// TwinCAT 3 PLC project PLC1
// ProgramVersion: 3.1.4026.23
// libraries:
//   Tc2_EtherCAT, * (Beckhoff Automation GmbH)
//   Tc2_Standard, * (Beckhoff Automation GmbH)
//   Tc2_System, * (Beckhoff Automation GmbH)
// project tree:
//   / PlcTask.TcTTO
//   POUs/ F_ConsumeTime.TcPOU, PRG_PLC1.TcPOU
// real-time tasks:
//   TASK PlcTask: cycle T#10ms, priority 20, ADS port 350
// variable links:
//   PLC1/PLC1 Instance <-> PLC2/PLC2 Instance
//     PlcTask Inputs/PRG_PLC1.FromPLC2 <-> PlcTask Outputs/PRG_PLC2.ToPLC_X
//     PlcTask Outputs/PRG_PLC1.ToPLC_X <-> PlcTask Inputs/PRG_PLC2.FromPLC1
//   PLC1/PLC1 Instance <-> PLC3/PLC3 Instance
//     PlcTask Inputs/PRG_PLC1.FromPLC3 <-> PlcTask Outputs/PRG_PLC3.ToPLC_X
//     PlcTask Outputs/PRG_PLC1.ToPLC_X <-> PlcTask Inputs/PRG_PLC3.FromPLC1
//   PLC2/PLC2 Instance <-> PLC3/PLC3 Instance
//     PlcTask Inputs/PRG_PLC2.FromPLC3 <-> PlcTask Outputs/PRG_PLC3.ToPLC_X
//     PlcTask Outputs/PRG_PLC2.ToPLC_X <-> PlcTask Inputs/PRG_PLC3.FromPLC2

CONFIGURATION PLC1
    RESOURCE PLC ON TwinCAT3
        TASK PlcTask(INTERVAL := T#10ms, PRIORITY := 20);
        PROGRAM PRG_PLC1 WITH PlcTask : PRG_PLC1;
    END_RESOURCE
END_CONFIGURATION

// ---- POUs/PRG_PLC1.TcPOU
PROGRAM PRG_PLC1
VAR
	ToPLC_X	  AT %Q* : UDINT;
	
	FromPLC2  AT %I*  :UDINT;
	FromPLC3  AT %I*  :UDINT;
END_VAR

F_ConsumeTime(5);
ToPLC_X := (ToPLC_X + 1) MOD 200;

END_PROGRAM

// ---- POUs/F_ConsumeTime.TcPOU
FUNCTION F_ConsumeTime
VAR_INPUT
	Us		:UDINT;
END_VAR
VAR
		tCurr, tEnd : T_DCTIME64;
END_VAR

tCurr := F_GetActualDcTime64();
tEnd  := tCurr + (Us * EC_DCTIME_TICKSPERMSEC64 / 1000);
WHILE (tCurr < tEnd) DO
	tCurr := F_GetActualDcTime64();
END_WHILE

END_FUNCTION
